{attribute 'qualified_only'}
VAR_GLOBAL
	logMessage : STRING(255) := 'No Message';
END_VAR

(* stored: Version 1.1.0.1, ProductVersion 3.1.4022.18
   GVL GVL: Id {9f0e5451-815c-45fc-b84a-c5d91136f9d8} *)
